// TIA Portal V18 export
DATA_BLOCK "Stacklight_DB"   // DB83
VERSION : 0.1
// stored: AutoNumber true, DBAccessibleFromOPCUA true, InstanceOfName Stacklight, InstanceOfType FB
"Stacklight"
   // VAR_INPUT
   //    Emergency : Bool;
   //    Mode : Int;
   //    RedIn : Bool;
   //    YellowIn : Bool;
   //    GreenIn : Bool;
   //    ReadyDevices : Bool;
   //    DoorOpen : Bool;
   //    Xvelocity : DInt;
   //    Yvelocity : DInt;
   //    MachineReadyPLC : Bool;
   //    MachineReadyNOAH : Bool;
   //    MachinePrintingPLC : Bool;
   //    MachinePrintingNOAH : Bool;
   //    MachineErrorPLC : Bool;
   //    MachineErrorNOAH : Bool;
   //    LED01 : Bool;
   //    LED02 : Bool;
   //    Maintenance : Int;
   // END_VAR
   // VAR_OUTPUT
   //    Status : Int;
   //    OutputColor : Int;
   //    StacklightCTRL01 : Bool;
   //    StacklightCTRL02 : Bool;
   // END_VAR
   // VAR_IN_OUT
   //    MachineConnectedNOAH : Bool;
   // END_VAR
   // VAR
   //    TriggerVelocityForMoving : DInt;
   //    GreenInternal : Bool;
   //    YellowInternal : Bool;
   //    RedInternal : Bool;
   //    ColorInternal : Int;
   //    MachineMovingInternal : Bool;
   //    MachineConnectedPLC : Bool;
   //    MachineConnectedInternal : Bool;
   // END_VAR
BEGIN
END_DATA_BLOCK
